FUNCTION Fal : LREAL
VAR_INPUT
	e:LREAL;
	alpha:LREAL;
	delta:LREAL;
END_VAR
VAR
	temp:LREAL;
END_VAR

//原点附近有连线性段的连续幂次函数
IF ABS(e) <= delta THEN
	Fal := e / EXPT(delta, alpha -1);
ELSE
	Fal := EXPT(ABS(e), alpha) * Sign(e);
END_IF
//temp := (Sign(e+delta) - Sign(e-delta)) / 2;
//Fal := e * temp / (EXPT(delta, 1 - alpha)) + EXPT(ABS(e), alpha) * Sign(e) * (1 - temp);

END_FUNCTION

(* stored: Version 1.1.0.1, ProductVersion 3.1.4024.11
   POU Fal: Id {0b2ee681-25be-4f41-b01f-4532847a1a77}, SpecialFunc None *)
